FUNCTION Sum : LREAL
VAR_INPUT
    var1 : LREAL;
    var2 : LREAL;
END_VAR
VAR
    total : LREAL;
END_VAR

// Body

END_FUNCTION

(* stored: Version 1.1.0.1, ProductVersion 3.1.4024.3
   POU Sum: Id {5ef86b57-8d8e-4047-bb1e-6f2aaafbe9aa}, SpecialFunc None *)
